// TIA Portal V19 export
TYPE "LEXCHANGETRAY_typeCellsInterface"
// stored: Access Published
   STRUCT
      monitor : "LEXCHANGETRAY_typeCellsMonitor";   // 电池信息
   END_STRUCT;
END_TYPE
